// TIA Portal V20 export
TYPE "type_emRelations_em4_SoftCam"
// stored: Access Published, Namespace Unit1
   STRUCT
      sideTapeFixStageAxisX : Struct
         pos00_wait : "LER_typeSoftCamPosition";
         pos01_load : "LER_typeSoftCamPosition";
         pos02_unload : "LER_typeSoftCamPosition";
         pos03_posistion : "LER_typeSoftCamPosition";
         pos04_posistion : "LER_typeSoftCamPosition";
         pos05_posistion : "LER_typeSoftCamPosition";
         pos06_posistion : "LER_typeSoftCamPosition";
         pos07_posistion : "LER_typeSoftCamPosition";
         pos08_posistion : "LER_typeSoftCamPosition";
         pos09_posistion : "LER_typeSoftCamPosition";
         pos10_posistion : "LER_typeSoftCamPosition";
         pos11_posistion : "LER_typeSoftCamPosition";
         pos12_posistion : "LER_typeSoftCamPosition";
         pos13_posistion : "LER_typeSoftCamPosition";
         pos14_posistion : "LER_typeSoftCamPosition";
         pos15_posistion : "LER_typeSoftCamPosition";
      END_STRUCT;
      sideTapeFixStageAxisC : Struct
         pos00_tape1 : "LER_typeSoftCamPosition";
         pos01_tape2 : "LER_typeSoftCamPosition";
         pos02_tape3 : "LER_typeSoftCamPosition";
         pos03_tape4 : "LER_typeSoftCamPosition";
         pos04_posistion : "LER_typeSoftCamPosition";
         pos05_posistion : "LER_typeSoftCamPosition";
         pos06_posistion : "LER_typeSoftCamPosition";
         pos07_posistion : "LER_typeSoftCamPosition";
         pos08_posistion : "LER_typeSoftCamPosition";
         pos09_posistion : "LER_typeSoftCamPosition";
         pos10_posistion : "LER_typeSoftCamPosition";
         pos11_posistion : "LER_typeSoftCamPosition";
         pos12_posistion : "LER_typeSoftCamPosition";
         pos13_posistion : "LER_typeSoftCamPosition";
         pos14_posistion : "LER_typeSoftCamPosition";
         pos15_posistion : "LER_typeSoftCamPosition";
      END_STRUCT;
      sideTapeAttachmentAxisX : Struct
         pos00_wait : "LER_typeSoftCamPosition";
         pos01_rightTapeGet : "LER_typeSoftCamPosition";
         pos02_leftTapeGet : "LER_typeSoftCamPosition";
         pos03_tape1Put : "LER_typeSoftCamPosition";
         pos04_tape2Put : "LER_typeSoftCamPosition";
         pos05_tape3Put : "LER_typeSoftCamPosition";
         pos06_tape4Put : "LER_typeSoftCamPosition";
         pos07_remainAttachLeft : "LER_typeSoftCamPosition";
         pos08_remainAttachRight : "LER_typeSoftCamPosition";
         pos09_tapePutZone : "LER_typeSoftCamPosition";
         pos10_posistion : "LER_typeSoftCamPosition";
         pos11_posistion : "LER_typeSoftCamPosition";
         pos12_posistion : "LER_typeSoftCamPosition";
         pos13_posistion : "LER_typeSoftCamPosition";
         pos14_posistion : "LER_typeSoftCamPosition";
         pos15_posistion : "LER_typeSoftCamPosition";
      END_STRUCT;
      sideTapeAttachmentAxisY : Struct
         Pos00_wait : "LER_typeSoftCamPosition";
         pos01_rightTapeGet : "LER_typeSoftCamPosition";
         pos02_leftTapeGet : "LER_typeSoftCamPosition";
         pos03_tape1Put : "LER_typeSoftCamPosition";
         pos04_tape2Put : "LER_typeSoftCamPosition";
         pos05_tape3Put : "LER_typeSoftCamPosition";
         pos06_tape4Put : "LER_typeSoftCamPosition";
         pos07_remainAttachLeft : "LER_typeSoftCamPosition";
         pos08_remainAttachRight : "LER_typeSoftCamPosition";
         pos09_noInterferenceZone : "LER_typeSoftCamPosition";
         pos10_posistion : "LER_typeSoftCamPosition";
         pos11_posistion : "LER_typeSoftCamPosition";
         pos12_posistion : "LER_typeSoftCamPosition";
         pos13_posistion : "LER_typeSoftCamPosition";
         pos14_posistion : "LER_typeSoftCamPosition";
         pos15_posistion : "LER_typeSoftCamPosition";
      END_STRUCT;
   END_STRUCT;
END_TYPE
